(* CODESYS project GVL_HMI.gvl.xml

Project tree, tasks and I/O mapping:
  global variables GVL_HMI
*)

// GVL_HMI
{attribute 'qualified_only'}
VAR_GLOBAL
	HMI : ST_HMI;
END_VAR
